TYPE TcaLaserDistanceSensorDataArrayEntry :
STRUCT
	x			: DINT;
	y			: DINT;
END_STRUCT
END_TYPE

(* stored: Version 1.1.0.1
   DUT TcaLaserDistanceSensorDataArrayEntry: Id {f65edd29-4a2a-49df-8602-69b9d89e747c} *)
